PROGRAM MAIN
VAR
	programIsRunning : USINT;
	
	hiveMQ_MQTT : HiveMQ_MQTT;
END_VAR

programIsRunning := programIsRunning + 1;

hiveMQ_MQTT();
// hiveMQ_MQTT.CyclicCode();

END_PROGRAM

(* stored: Version 1.1.0.1
   POU MAIN: Id {9cdf4ae1-9b2e-4987-84f5-d15c56852726}, SpecialFunc None *)
